{region '#Template'}
	{attribute 'Category' := 'General'}
	{attribute 'Version' := '0.0.1.0'}
	{attribute 'Tags' := 'General, Cabinet, Control cabinet, Acknowledgement'}
	{attribute 'Description' := 'Schaltschrank Quittierung	// Control cabinet acknowledgement'}
{endregion}
FUNCTION_BLOCK FB_BA_ControlCabinetBasic EXTENDS FB_BA_View
VAR
	// By default, the entire project structure can be acknowledged.
	// There may be constellations (e.g. multiple control cabinets) where only one part of the project structure (e.g. multiple buildings) has to be acknowledged.
	// > In this case separete parts can be assigned here: 
	iAckView1				: I_BA_View;
	iAckView2				: I_BA_View;
	iAckView3				: I_BA_View;
END_VAR
VAR_INPUT CONSTANT
	LampFault				: FB_BA_ActuatorCmd;		
	AckButton				: FB_BA_CombinationBI_BV;													
	RstHw					: FB_BA_ActuatorCmd;														
END_VAR
VAR				
	bIsDisturbed			: BOOL;
	bHasUnackEvent			: BOOL;
	bBlink					: BOOL;
	tAlmLampImpuls			: FB_BA_Blink;						
	tpResetHw				: TP;	
	rtrigRstSwi				: R_TRIG;
	bTrigRstSwi				: BOOL;
	rtrigRstButton			: R_TRIG;
	bTrigRstButton			: BOOL;	
END_VAR

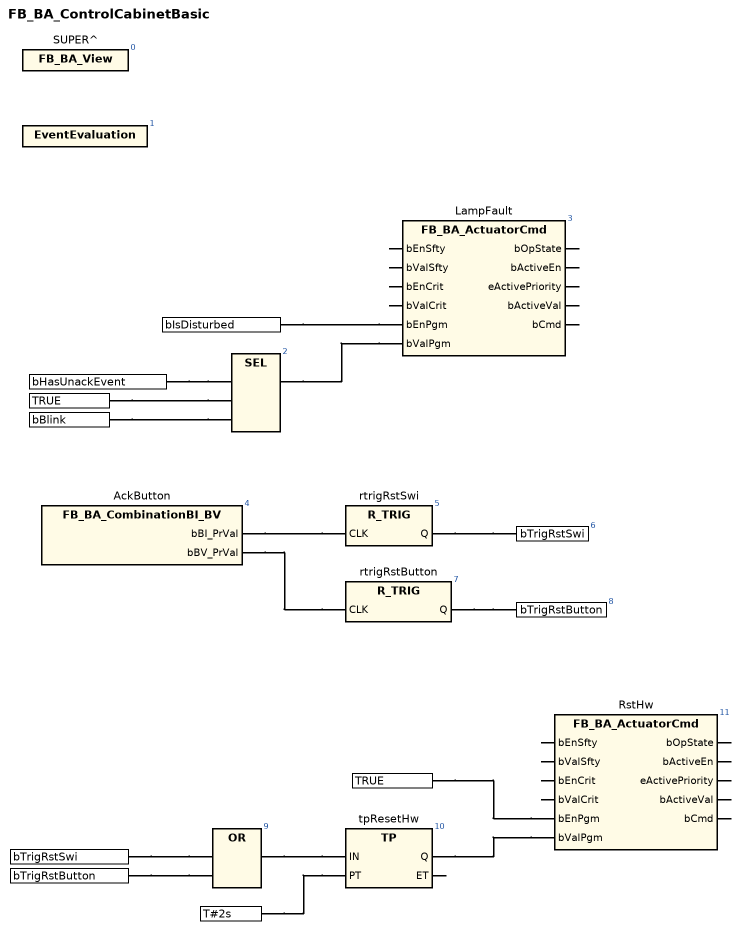
SUPER^(); // FB_BA_View
EventEvaluation();
LampFault(bEnPgm := bIsDisturbed, bValPgm := SEL(bHasUnackEvent, TRUE, bBlink)); // FB_BA_ActuatorCmd
AckButton(); // FB_BA_CombinationBI_BV
rtrigRstSwi(CLK := AckButton.bBI_PrVal); // R_TRIG
bTrigRstSwi := rtrigRstSwi.Q;
rtrigRstButton(CLK := AckButton.bBV_PrVal); // R_TRIG
bTrigRstButton := rtrigRstButton.Q;
tpResetHw(IN := bTrigRstSwi OR bTrigRstButton, PT := T#2s); // TP
RstHw(bEnPgm := TRUE, bValPgm := tpResetHw.Q); // FB_BA_ActuatorCmd

METHOD PRIVATE Ack
VAR_INPUT
	iView			: I_BA_View;
END_VAR
IF (iView <> 0) THEN
	iView.AcknowledgeObjectsPLC := (bTrigRstSwi) OR (bTrigRstButton);	
END_IF
END_METHOD

METHOD PRIVATE EventEvaluation
VAR
	_iView			: I_BA_View;
END_VAR
bIsDisturbed := FALSE;
bHasUnackEvent := FALSE;

IF (iAckView1 = 0) AND (iAckView2 = 0) AND (iAckView3 = 0) THEN
	// Treat project structure via root-object:
	Ack(BA_Globals.Top);
	GetErrors(BA_Globals.Top);
ELSE
	// Treat each defined object:
	Ack(iAckView1);
	GetErrors(iAckView1);
	
	Ack(iAckView2);
	GetErrors(iAckView2);
	
	Ack(iAckView3);
	GetErrors(iAckView3);
END_IF

// Generate alarm lamp impulse:
tAlmLampImpuls();

bBlink := tAlmLampImpuls.bQ;
END_METHOD

METHOD FB_init : BOOL
VAR_INPUT
	bInitRetains : BOOL; // if TRUE, the retain variables are initialized (warm start / cold start)
	bInCopyCode : BOOL;  // if TRUE, the instance afterwards gets moved into the copy code (online change)
END_VAR
LampFault.iParent							:= THIS^;
LampFault.iLabel							:= LblCmpGeneral.ControlCabinet_LampFault;			
LampFault.sObjectName						:= '{Idx=01}';
LampFault.eDPADMode							:= E_BA_DPADMode.eInclude;																						
LampFault.Cmd.iLabel						:= LblCmpGeneral.ControlCabinet_LampFault_Cmd;			
LampFault.Cmd.sObjectName					:= '{Idx=01}';	
LampFault.Cmd.ePolarity						:= E_BA_Polarity.eNormal;
LampFault.Cmd.eFeedbackPolarity				:= E_BA_Polarity.eNormal;
LampFault.Cmd.eOverriddenPolarity			:= E_BA_Polarity.eReverse;
LampFault.Cmd.sActiveText 					:= Texts.txtOn;
LampFault.Cmd.sInactiveText 				:= Texts.txtOff;
LampFault.Cmd.nEventClassID					:= EventClasses.DisturbanceExtended;
LampFault.Cmd.aEventTransitionText[1]		:= Texts.txtDisturb;
LampFault.Cmd.aEventTransitionText[2]		:= Texts.txtNone;
LampFault.Cmd.aEventTransitionText[3]		:= Texts.txtNormal;
LampFault.Cmd.bEventDetectionEnable			:= TRUE;
LampFault.Cmd.eEnPlantLock					:= E_BA_LockPriority.eNoLock;	

AckButton.iParent							:= THIS^;		
AckButton.iLabel 							:= LblCmpGeneral.ControlCabinet_AckButton;	
AckButton.sObjectName						:= '{Idx=01}';
AckButton.eDPADMode							:= E_BA_DPADMode.eInclude;																						
AckButton.Input.iLabel						:= LblCmpGeneral.ControlCabinet_AckButton_Input;
AckButton.Input.ePolarity					:= E_BA_Polarity.eNormal;
AckButton.Value.iLabel						:= LblCmpGeneral.ControlCabinet_AckButton_Value;
AckButton.Value.eToggleMode 				:= E_BA_ToggleMode.ePushButton;									

RstHw.iParent								:= THIS^;
RstHw.iLabel								:= LblCmpGeneral.ControlCabinet_RstHw;			
RstHw.sObjectName							:= '{Idx=02}';
RstHw.eDPADMode								:= E_BA_DPADMode.eInclude;																						
RstHw.Cmd.iLabel							:= LblCmpGeneral.ControlCabinet_RstHw_Cmd;			
RstHw.Cmd.sObjectName						:= '{Idx=01}';	
RstHw.Cmd.ePolarity							:= E_BA_Polarity.eNormal;
RstHw.Cmd.eFeedbackPolarity					:= E_BA_Polarity.eNormal;
RstHw.Cmd.eOverriddenPolarity				:= E_BA_Polarity.eReverse;
RstHw.Cmd.sActiveText 						:= Texts.txtOn;
RstHw.Cmd.sInactiveText 					:= Texts.txtOff;
RstHw.Cmd.nEventClassID						:= EventClasses.DisturbanceExtended;
RstHw.Cmd.aEventTransitionText[1]			:= Texts.txtDisturb;
RstHw.Cmd.aEventTransitionText[2]			:= Texts.txtNone;
RstHw.Cmd.aEventTransitionText[3]			:= Texts.txtNormal;
RstHw.Cmd.bEventDetectionEnable				:= TRUE;
RstHw.Cmd.eEnPlantLock						:= E_BA_LockPriority.eNoLock;	

tAlmLampImpuls.bEn							:=	TRUE; 
tAlmLampImpuls.nTiOn						:=	800;
tAlmLampImpuls.nTiOff						:=	800;
END_METHOD

METHOD PRIVATE GetErrors
VAR_INPUT
	iView			: I_BA_View;
END_VAR
VAR
	iTemp			: INT;
	fbEvents		: REFERENCE TO FB_BA_EventIndicator;
END_VAR
IF (iView <> 0) THEN
	fbEvents REF= iView.ActiveEvents;
	
	FOR iTemp := E_BA_EventType.First TO E_BA_EventType.Last DO
		IF (fbEvents.aEventsPerIconImage[iTemp].nCount > 0) THEN
			bIsDisturbed := TRUE;
			
			CASE (fbEvents.aEventsPerIconImage[iTemp].eMostPriorisedState) OF
				E_BA_EventIconState.ePresent,
				E_BA_EventIconState.eGone:
					bHasUnackEvent := TRUE;
			END_CASE
		END_IF
	END_FOR
END_IF
END_METHOD

METHOD PROTECTED Reset
VAR_INPUT
	bUnregister			: BOOL			:= FALSE;
END_VAR
iAckView1 := 0;
iAckView2 := 0;
iAckView3 := 0;

SUPER^.Reset(bUnregister);
END_METHOD

END_FUNCTION_BLOCK

(* stored: Version 1.1.0.1, ProductVersion 3.1.4024.6
   POU FB_BA_ControlCabinetBasic: Id {550107ee-d771-4323-800a-04af4104ef22}, SpecialFunc None
   Folder [Private]: Id {024b046a-664d-49d2-bb07-97be0eadde0d}
   Folder [Protected] Management: Id {85912088-ad90-47de-97a7-570e488812bc}
   Method Ack: Id {af109ea4-070e-4e58-b5ce-40236a2c408d}
   Method EventEvaluation: Id {a7916a83-24ce-43a5-9205-f7f86645c89c}
   Method FB_init: Id {12d1fc59-1c6e-471b-895f-17582d0de6f1}
   Method GetErrors: Id {7d4cdfdd-7941-4230-96bd-fd54056feeea}
   Method Reset: Id {4b7e996f-2b2c-4a34-8b96-5546044e48cc} *)
